SUBAPPLICATION mapping_Softkeys (* Subapplication Type *)
  (* Standard: 61499-2 *)
  (* Version 1.0, 2023-01-29, Franz *)
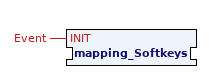
  EVENT_INPUT
    INIT;
  END_EVENT
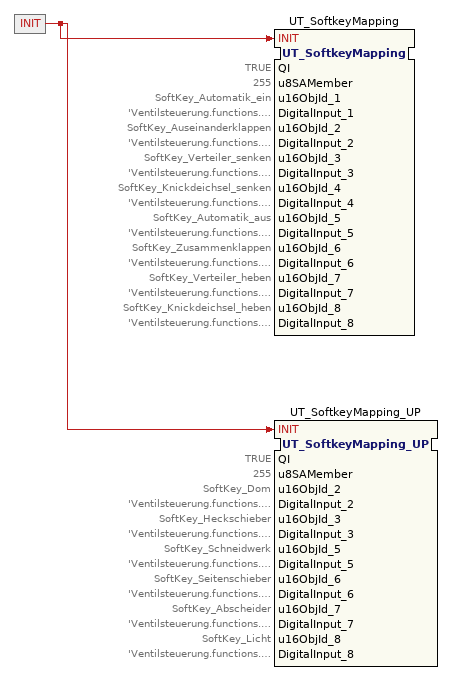
  FBS
    UT_SoftkeyMapping : UT_SoftkeyMapping(QI := TRUE, u8SAMember := 255, u16ObjId_1 := SoftKey_Automatik_ein, DigitalInput_1 := 'Ventilsteuerung.functions.Automatik.ein.SoftKey', u16ObjId_2 := SoftKey_Auseinanderklappen, DigitalInput_2 := 'Ventilsteuerung.functions.Klappen.SoftKey_heben.IX', u16ObjId_3 := SoftKey_Verteiler_senken, DigitalInput_3 := 'Ventilsteuerung.functions.Verteiler.SoftKey_senken.IX', u16ObjId_4 := SoftKey_Knickdeichsel_senken, DigitalInput_4 := 'Ventilsteuerung.functions.Knickdeichsel.SoftKey_senken.IX', u16ObjId_5 := SoftKey_Automatik_aus, DigitalInput_5 := 'Ventilsteuerung.functions.Automatik.aus.SoftKey', u16ObjId_6 := SoftKey_Zusammenklappen, DigitalInput_6 := 'Ventilsteuerung.functions.Klappen.SoftKey_senken.IX', u16ObjId_7 := SoftKey_Verteiler_heben, DigitalInput_7 := 'Ventilsteuerung.functions.Verteiler.SoftKey_heben.IX', u16ObjId_8 := SoftKey_Knickdeichsel_heben, DigitalInput_8 := 'Ventilsteuerung.functions.Knickdeichsel.SoftKey_heben.IX');
    UT_SoftkeyMapping_UP : UT_SoftkeyMapping_UP(QI := TRUE, u8SAMember := 255, u16ObjId_2 := SoftKey_Dom, DigitalInput_2 := 'Ventilsteuerung.functions.Dom.SoftKey_UP.IE', u16ObjId_3 := SoftKey_Heckschieber, DigitalInput_3 := 'Ventilsteuerung.functions.Heckschieber.SoftKey_UP.IE', u16ObjId_5 := SoftKey_Schneidwerk, DigitalInput_5 := 'Ventilsteuerung.functions.Schneidwerk.SoftKey_UP.IE', u16ObjId_6 := SoftKey_Seitenschieber, DigitalInput_6 := 'Ventilsteuerung.functions.Seitenschieber.SoftKey_UP.IE', u16ObjId_7 := SoftKey_Abscheider, DigitalInput_7 := 'Ventilsteuerung.functions.Abscheider.SoftKey_UP.IE', u16ObjId_8 := SoftKey_Licht, DigitalInput_8 := 'Ventilsteuerung.functions.Licht.SoftKey_UP.IE');
  END_FBS
  EVENT_CONNECTIONS
    INIT TO UT_SoftkeyMapping.INIT;
    INIT TO UT_SoftkeyMapping_UP.INIT;
  END_CONNECTIONS
END_SUBAPPLICATION
